FUNCTION F_ChkSettingUserLevel : BOOL
VAR_INPUT
	eLevel		: E_User_Level;
END_VAR
VAR_IN_OUT
	stSetting 	: ST_Data_Item;
END_VAR
VAR_OUTPUT
	stInfo 		: ST_Text;
END_VAR

F_ChkSettingUserLevel := FALSE;

IF (eUserLevel < stSetting.eUserLevel) THEN
	stInfo.wsName := "incorrect user level";
	stInfo.wsNameId := "incorrectuserlevel";
	RETURN;
END_IF

IF(stSetting.eDataType = E_DataType.eDataType_None)	THEN
	stInfo.wsName := "incorrect type";
	stInfo.wsNameId := "incorrecttype";
	RETURN;					
END_IF

F_ChkSettingUserLevel := TRUE;

END_FUNCTION

(* stored: Version 1.1.0.1, ProductVersion 3.1.4024.12
   POU F_ChkSettingUserLevel: Id {16f240dc-b7a0-4c79-a8fc-a56924f74a86}, SpecialFunc None *)
